// SIMATIC STEP 7 (V5.x) project ZEn01_11_STEP7__Com_SFC1
// program: ProgrammClient(MPI=10)
// program: ProgrammServer(MPI=12)
// program: ProgrammServer(MPI=15)

SYMBOL_TABLE
"Data_X_PUT"	DB 1	DB 1
"Data_X_GET"	DB 2	DB 2
"Data_X_SEND"	DB 3	DB 3
"Modify Values"	FC 1	FC 1
"Communication(send)"	FC 10	FC 10
"CYCL_EXC"	OB 1	OB 1	// Cycle Execution
"CYC_INT5"	OB 35	OB 35	// Cyclic Interrupt 5
"COMPLETE RESTART"	OB 100	OB 100	// Complete Restart
"X_SEND"	SFC 65	SFC 65
"X_RCV"	SFC 66	SFC 66
"X_GET"	SFC 67	SFC 67
"X_PUT"	SFC 68	SFC 68
"X_ABORT"	SFC 69	SFC 69
"I_GET"	SFC 72	SFC 72
"I_PUT"	SFC 73	SFC 73
"I_ABORT"	SFC 74	SFC 74
END_SYMBOL_TABLE

FUNCTION "Modify Values" : VOID	// FC 1
TITLE = Function for Generating a Modifiable Date
AUTHOR : SIEMENS
VERSION : 1.0
BEGIN
NETWORK
TITLE = Incrementing and Saving a Value
      L     MD 60;
      L     1;
      +D;
      T     MD 60;
      T     DB1.DBD 0;	//Save the variables to be sent in a double word
      T     DB3.DBD 0;
END_FUNCTION

FUNCTION "Communication(send)" : VOID	// FC 10
TITLE = Communicating with Both Servers
AUTHOR : SIEMENS
VERSION : 1.0
BEGIN
NETWORK
TITLE = Communicating with Server MPI 15
//Scan to see whether the SFCs X_PUT, X_GET, and X_SEND have communicated with 
//server MPI 15
      A     M 100.6;	//SFC X_PUT: Communication finished?
      A     M 101.6;	//SFC X_GET: Communication finished?
      A     M 102.6;	//SFC X_SEND: Communication finished?
      JC    net2;	//Jump to communication with server MPI 12
//                                        if the condtion is fulfilled. 
//Query which SFC is currently active?
      L     MW 50;	//SFC X_PUT active?
      L     1;
      ==I;
      JC    m001;	//Jump to SFC X_PUT
      L     MW 50;	//SFC X_GET active?
      L     2;
      ==I;
      JC    m002;	//Jump to SFC X_GET
      L     MW 50;	//SFC X_SEND active?
      L     3;
      ==I;
      JC    m003;	//Jump to SFC X_SEND
      BEU;
m001: CALL  "X_PUT" (
           REQ                      := M 100.2,
           CONT                     := M 100.3,
           DEST_ID                  := W#16#F,
           VAR_ADDR                 := "Data_X_PUT".Array10Bytes,
           SD                       := "Data_X_PUT".Array10Bytes,
           RET_VAL                  := MW 130,
           BUSY                     := M 100.4);	//Call X_PUT block / Transfer data (Yes/No)? / Maintain connection (Yes/No)? / Address of receiver / Address within communication partner / Send data 10 bytes (DB1) / Status display, negative if an error occurs / SFC active?
//Edge evaluation: Is communication with the falling edge of the BUSY bit
//finished?
      A     M 100.4;
      FN    M 100.5;
      S     M 100.6;	//Set memory bit: X_PUT is finished.
      JC    m004;	//Jump to increment the communication memory bit
      BEU;
m002: CALL  "X_GET" (
           REQ                      := M 101.2,
           CONT                     := M 101.3,
           DEST_ID                  := W#16#F,
           VAR_ADDR                 := "Data_X_GET".DoubleWord,
           RET_VAL                  := MW 132,
           BUSY                     := M 101.4,
           RD                       := "Data_X_GET".DoubleWord);	//Call X_SEND block / Transfer data (Yes/No)? / Maintain connection (Yes/No)? / Address of receiver / Address of variable in communication partner / Status display, negative if an error occurs / SFC active? / Pointer to address to which receive data are written
//Edge evaluation: Is communication with the falling edge of the BUSY bit
//finished?
      A     M 101.4;
      FN    M 101.5;
      S     M 101.6;	//Set memory bit: X_GET is finished.
      JC    m005;	//Jump to increment the communication counter
      BEU;
m003: CALL  "X_SEND" (
           REQ                      := M 102.2,
           CONT                     := M 102.3,
           DEST_ID                  := W#16#F,
           REQ_ID                   := DW#16#3,
           SD                       := "Data_X_SEND".Array3Words,
           RET_VAL                  := MW 134,
           BUSY                     := M 102.4);	//Call X_SEND block / Transfer data (Yes/No)? / Maintain connection (Yes/No)? / Address of receiver / Job number 3 / Send data 3 words (DB3) / Status display / SFC active?
//Edge evaluation: Is communication with the falling edge of the BUSY bit
//finished?
      A     M 102.4;
      FN    M 102.5;
      S     M 102.6;	//Set memory bit: X_SEND is finished.
      JC    m006;	//Jump to increment the communication counter
      BEU;
//In the following section, the communication counter is incremented following communication. 
m004: L     2;	//Increment on executing X_PUT
      T     MW 50;
      CALL  "Modify Values";	//The values in the variables are incremented
      BEU;
m005: L     3;	//Increment on executing X_GET
      T     MW 50;
      CALL  "Modify Values";	//The values in the variables are incremented
      BEU;
m006: L     1;	//Increment on executing X_SEND
      T     MW 50;
      CALL  "Modify Values";	//The values in the variables are incremented
NETWORK
TITLE = Communicating with Server MPI 12
//Query which SFC is currently active
net2: L     MW 52;	//SFC X_ABORT active?
      L     1;
      ==I;
      JC    m007;	//Jump to SFC X_ABORT
      L     MW 52;	//SFC X_SEND active?
      L     2;
      ==I;
      JC    m008;	//Jump to SFC X_SEND
      L     MW 52;	//SFC X_ABORT active?
      L     3;
      ==I;
      JC    m009;	//Jump to SFC X_ABORT
      BEU;
//In the following section of this network, the SFC X_ABORT is called to disconnect the 
//connection to the server MPI 15 which was established in network 1.
//The connection resource for SFC X_SEND in this network is available for this.
m007: CALL  "X_ABORT" (
           REQ                      := M 104.2,
           DEST_ID                  := W#16#F,
           RET_VAL                  := MW 136,
           BUSY                     := M 104.4);	//Call to abort connection to CPU-MPI 15 / Abort connection to CPU MPI address 15? / MPI address 15 / Return value of SFC / SFC active?
//Edge evaluation: Has the connection been aborted with the falling edge of the BUSY bit?
      A     M 104.4;
      FN    M 104.5;
      JC    m010;	//Jump to increment the communication memory word
      BEU;
//In the following section of this network, the SFC X_SEND is called to communicate 
//with the server MPI 12.
m008: CALL  "X_SEND" (
           REQ                      := M 105.2,
           CONT                     := M 105.3,
           DEST_ID                  := W#16#C,
           REQ_ID                   := DW#16#2,
           SD                       := "Data_X_PUT".Array10Bytes,
           RET_VAL                  := MW 138,
           BUSY                     := M 105.4);	//Call SFC X_SEND / Start data exchange? / Maintain connection following communication? / MPI address 12 / Job number 2 / Variable to be sent / Return value for error evaluation / SFC active?
//Edge evaluation: Is communication with the falling edge of the BUSY bit
//finished?
      A     M 105.4;
      FN    M 105.5;
      JC    m011;	//Jump to increment the communication memory word
      BEU;
//In the following section of this network, the SFC X_ABORT is called to disconnect the 
//connection to the server MPI 12 which was established in this network by SFC X_SEND.
//The connection resource for the SFCs in network 1 then becomes available again.
m009: CALL  "X_ABORT" (
           REQ                      := M 106.2,
           DEST_ID                  := W#16#C,
           RET_VAL                  := MW 140,
           BUSY                     := M 106.4);	//Call to abort connection to CPU MPI 12 / Abort connection to CPU MPI address 12? / MPI address 12
//Edge evaluation: Has the connection been aborted with the falling edge of the BUSY bit?
      A     M 106.4;
      FN    M 106.5;
      JC    m012;	//Jump to increment the communication memory word
      BEU;
//In the following section, the communication counter is incremented after an SFC has been 
//executed.
m010: L     2;	//Increment after executing X_ABORT with server MPI 15
      T     MW 52;
      BEU;
m011: L     3;	//Increment after executing X_SEND
      T     MW 52;
      BEU;
m012: L     1;	//Increment after executing X_ABORT with server MPI 12
      T     MW 52;
//Reset the memory bits in the first network: The SFC must have finished communicating 
//before the SFCs can be called again from the first network.
      CLR;
      =     M 100.6;	//Reset the memory bit: SFC X_PUT has been executed
      =     M 101.6;	//Reset the memory bit: SFC X_GET has been executed
      =     M 102.6;	//Reset the memory bit: SFC X_SEND has been executed
END_FUNCTION

DATA_BLOCK "Data_X_PUT"	// DB 1
AUTHOR : SIEMENS
VERSION : 1.0
  STRUCT
   Array10Bytes : ARRAY  [1 .. 10 ] OF //Array of 10 bytes
   BYTE  := 5 (B#16#10) , 5 (B#16#10) ;
  END_STRUCT ;	
BEGIN
   Array10Bytes[1] := B#16#10;
   Array10Bytes[2] := B#16#10;
   Array10Bytes[3] := B#16#10;
   Array10Bytes[4] := B#16#10;
   Array10Bytes[5] := B#16#10;
   Array10Bytes[6] := B#16#10;
   Array10Bytes[7] := B#16#10;
   Array10Bytes[8] := B#16#10;
   Array10Bytes[9] := B#16#10;
   Array10Bytes[10] := B#16#10;
END_DATA_BLOCK

DATA_BLOCK "Data_X_GET"	// DB 2
AUTHOR : SIEMENS
VERSION : 1.0
  STRUCT
   DoubleWord : DWORD  := DW#16#2D;	//Double word
  END_STRUCT ;	
BEGIN
   DoubleWord := DW#16#2D;
END_DATA_BLOCK

DATA_BLOCK "Data_X_SEND"	// DB 3
AUTHOR : SIEMENS
VERSION : 1.0
  STRUCT
   Array3Words : ARRAY  [1 .. 3 ] OF //Array of 3 words
   WORD  := 3 (W#16#3) ;
  END_STRUCT ;	
BEGIN
   Array3Words[1] := W#16#3;
   Array3Words[2] := W#16#3;
   Array3Words[3] := W#16#3;
END_DATA_BLOCK

ORGANIZATION_BLOCK "CYCL_EXC"	// OB 1
TITLE = Cyclically Processing Program
AUTHOR : SIEMENS
VERSION : 1.0
VAR_TEMP
  OB1_EV_CLASS : BYTE ;	//Bits 0 to 3 = 1 (incoming event), bits 4 to 7 = 1 (event class 1)
  OB1_SCAN_1 : BYTE ;	//1 (Cold restart scan 1 of OB1), 3 Scan 2-n of OB 1)
  OB1_PRIORITY : BYTE ;	//1 (Priority of 1 is lowest)
  OB1_OB_NUMBR : BYTE ;	//1 (Organization block 1, OB1)
  OB1_RESERVED_1 : BYTE ;	//Reserved for system
  OB1_RESERVED_2 : BYTE ;	//Reserved for system
  OB1_PREV_CYCLE : INT ;	//Cycle time of previous OB1 scan (milliseconds)
  OB1_MIN_CYCLE : INT ;	//Minimum cycle time of OB1 (milliseconds)
  OB1_MAX_CYCLE : INT ;	//Maximum cycle time of OB1 (milliseconds)
  OB1_DATE_TIME : DATE_AND_TIME ;	//Date and time OB1 started
END_VAR
BEGIN
NETWORK
TITLE = Default Settings of the SFC Parameters
//********************************************************************************
//********************
//General Description of the Communication Procedures of this Client CPU
//********************************************************************************
//********************
//
//Three variables are exchanged between this client station ("S7-300 Client MPI 
//10") and the two 
//server stations ("S7-300 Server MPI 12" and "S7-300 Server MPI 15").
//The variable "X_PUT-1".Feld10byte is sent to server MPI 15 with the SFC X_PUT 
//and to server MPI 10 
//with the SFC X_SEND. You only require one connection resource in order to 
//communicate with the two 
//different servers, because the connections are disconnected with the SFC 
//X_ABORT between communication  
//procedures. In this way, connection resources for communication with other MPI 
//subnet partners are 
//not occupied unnecessarily. The variable "X_GET-1".Doppelwort is read out from 
//the server MPI 15 
//with the SFC X_GET and stored in a variable of the same name in the client.
//The variable "X_SEND-1".Feld3Worte is written by the client to a variable of 
//the same name on the 
//server with the SFC X_SEND.
//The variables can be found in DBs 1 to 3 on both the client and the server 
//side. 
//The connection between the communicating CPUs is established the first time an 
//SFC is called
//and then maintained until the connection is disconnected and then established 
//again for 
//the next communication partner (only one connection resource is required).
//The SFCs are called by OB35 using a timer in order to make them independent of 
//the  
//scan cycle time of OB1 in the client and the server CPU.
//The timers for the OB calls are preset when the CPU is configured.
//In this CPU, OB35 is called every 100 ms (default), and this means that the 
//various SFCs are also 
//called every 100 ms (max.). 
//Once data exchange is complete, the data are changed in the variables in order 
//to show that  
//data have been received. If there is an error in the communication, and no data 
//are
//sent, the data in the receiver will not change. 
//If the receive data are continually changing, this means that data exchange is 
//taking place.
//
//Note:
//The memory words in which the RET_VALS of the SFCs are entered should be 
//evaluated while the  
//program is running. If an SFC registers an error value, the SFC calls which are 
//locked 
//in this example with the falling edge of the BUSY output may be correctly 
//executed. However,  
//no data will have been sent. If an SFC call is correctly executed and its 
//RET_VAL still 
//registers an error code, it is essential that you forward an error message to 
//this effect to 
//the user. As soon as the RET_VAL of an SFC becomes negative, this signals that 
//an error has
//occurred and that data may have been lost.
//
//Memory words in which the RET_VALs are entered:
//MW130, MW132, MW134, MW136, MW138, MW140
//
//The above note was not taken into account in this programming example, since 
//error messages 
//which may occur cannot be converted to corresponding messages (alarms which 
//appear on the device) 
//until a real control program is run.
NETWORK
TITLE = Presetting Communication
//By setting the following three memory bits, you can ensure that the connection 
//between 
//the communication partners is retained following each SFC call.
      SET;
      =     M 100.3;	//Connection should be maintained after SFC call 
      =     M 101.3;	//Connection should be maintained after SFC call
      =     M 102.3;	//Connection should be maintained after SFC call 
      =     M 105.3;	//Connection should be maintained after SFC call 
//Set start memory bit of SFC
      SET;
      =     M 100.2;	//SFC X_PUT 
      =     M 101.2;	//SFC X_GET
      =     M 102.2;	//SFC X_SEND
      =     M 104.2;	//SFC X_ABORT
      =     M 105.2;	//SFC X_SEND
      =     M 106.2;	//SFC X_ABORT
END_ORGANIZATION_BLOCK

ORGANIZATION_BLOCK "CYC_INT5"	// OB 35
TITLE = Block Call Timer-Controlled Every 100 ms
AUTHOR : SIEMENS
VERSION : 1.0
VAR_TEMP
  OB35_EV_CLASS : BYTE ;	//Bits 0 to 3 = 1 (incoming event), bits 4 to 7 = 1 (event class 1)
  OB35_STRT_INF : BYTE ;	//16#36 (OB35 has started)
  OB35_PRIORITY : BYTE ;	//11 (Priority of 1 is lowest)
  OB35_OB_NUMBR : BYTE ;	//35 (Organization block 35, OB35)
  OB35_RESERVED_1 : BYTE ;	//Reserved for system
  OB35_RESERVED_2 : BYTE ;	//Reserved for system
  OB35_PHASE_OFFSET : WORD ;	//Phase offset (ms)
  OB35_RESERVED_3 : INT ;	//Reserved for system
  OB35_EXC_FREQ : INT ;	//Frequency of execution (ms)
  OB35_DATE_TIME : DATE_AND_TIME ;	//Date and time OB35 started
END_VAR
BEGIN
NETWORK
TITLE =
      CALL  "Communication(send)";	//Call communication with servers
END_ORGANIZATION_BLOCK

ORGANIZATION_BLOCK "COMPLETE RESTART"	// OB 100
AUTHOR : SIEMENS
VERSION : 1.0
VAR_TEMP
  OB100_EV_CLASS : BYTE ;	//16#13, Event class 1, entering event state, event logged in diagnostic buffer
  OB100_STRTUP : BYTE ;	//16#81/82/83/84 Method of startup
  OB100_PRIORITY : BYTE ;	//27 (Priority of 1 is lowest)
  OB100_OB_NUMBR : BYTE ;	//100 (Organization block 100, OB100)
  OB100_RESERVED_1 : BYTE ;	//Reserved for system
  OB100_RESERVED_2 : BYTE ;	//Reserved for system
  OB100_STOP : WORD ;	//Event that caused CPU to stop (16#4xxx)
  OB100_STRT_INFO : DWORD ;	//Information on how system started
  OB100_DATE_TIME : DATE_AND_TIME ;	//Date and time OB100 started
END_VAR
BEGIN
NETWORK
TITLE = Initial Value Assignment
      L     1;	//Start value for communication counter
//Communication counter for data exchange with the station "S7-300 Server MPI 15" 
      T     MW 50;
//Communication counter for data exchange with the station "S7-300 Server MPI 12" 
      T     MW 52;
END_ORGANIZATION_BLOCK

SYMBOL_TABLE
"Communication(receive)"	FC 20	FC 20
"CYCL_EXC"	OB 1	OB 1	// Cycle Execution
"CYC_INT5"	OB 35	OB 35	// Cyclic Interrupt 5
"COMPLETE RESTART"	OB 100	OB 100	// Complete Restart
"X_SEND"	SFC 65	SFC 65
"X_RCV"	SFC 66	SFC 66
"X_GET"	SFC 67	SFC 67
"X_PUT"	SFC 68	SFC 68
"X_ABORT"	SFC 69	SFC 69
"I_GET"	SFC 72	SFC 72
"I_PUT"	SFC 73	SFC 73
"I_ABORT"	SFC 74	SFC 74
END_SYMBOL_TABLE

FUNCTION "Communication(receive)" : VOID	// FC 20
AUTHOR : SIEMENS
VERSION : 1.0
VAR_TEMP
  NIL_PTR : ANY ;	//NIL pointer, required in order to discard data
END_VAR
BEGIN
NETWORK
TITLE = Timer-Controlled Call of the X_RCV Block
//In this block, the SFC X_RCV is called every 10 ms using a timer.
//
//If the receive data are not evaluated for any reason, they must be 
//removed from the receive buffer and written to a NIL pointer.
//The following section of this network contains the branch instruction which
//determines whether the data are received or discarded.
//
      JU    add;	//Jump to accept the receive data
//    SPA   disc                        //Jump to discard the receive data
      BEU;
add:  SET;	//Set the accept memory bit
      =     M 100.2;
      CALL  "X_RCV" (
           EN_DT                    := M 100.2,
           RET_VAL                  := MW 132,
           REQ_ID                   := MD 120,
           NDA                      := M 101.5,
           RD                       := P#M 100.0 BYTE 10);	//Call receive SFC to accept the data / Accept data? / Return value / Job number / Receive new data? / Data area to which the receive data are added
NETWORK
TITLE = Discarding the Receive Data
//disc: NOP   1                         //This line must be included if the 
//receive data are to be 
//                                        discarded with the NIL pointer.
// (network holds code this reader does not know; not shown)
END_FUNCTION

ORGANIZATION_BLOCK "CYCL_EXC"	// OB 1
VERSION : 0.1
VAR_TEMP
  OB1_EV_CLASS : BYTE ;	//Bits 0-3 = 1 (Coming event), Bits 4-7 = 1 (Event class 1)
  OB1_SCAN_1 : BYTE ;	//1 (Cold restart scan 1 of OB 1), 3 (Scan 2-n of OB 1)
  OB1_PRIORITY : BYTE ;	//1 (Priority of 1 is lowest)
  OB1_OB_NUMBR : BYTE ;	//1 (Organization block 1, OB1)
  OB1_RESERVED_1 : BYTE ;	//Reserved for system
  OB1_RESERVED_2 : BYTE ;	//Reserved for system
  OB1_PREV_CYCLE : INT ;	//Cycle time of previous OB1 scan (milliseconds)
  OB1_MIN_CYCLE : INT ;	//Minimum cycle time of OB1 (milliseconds)
  OB1_MAX_CYCLE : INT ;	//Maximum cycle time of OB1 (milliseconds)
  OB1_DATE_TIME : DATE_AND_TIME ;	//Date and time OB1 started
END_VAR
BEGIN
// (block stored without names or comments; labels and parameter names are numbered)
END_ORGANIZATION_BLOCK

ORGANIZATION_BLOCK "CYC_INT5"	// OB 35
TITLE = Call Every 100 ms
AUTHOR : SIEMENS
VERSION : 1.0
VAR_TEMP
  OB35_EV_CLASS : BYTE ;	//Bits 0 to 3 = 1 (incoming event), bits 4 to 7 = 1 (event class 1)
  OB35_STRT_INF : BYTE ;	//16#36 (OB35 has started)
  OB35_PRIORITY : BYTE ;	//11 (Priority of 1 is lowest)
  OB35_OB_NUMBR : BYTE ;	//35 (Organization block 35, OB35)
  OB35_RESERVED_1 : BYTE ;	//Reserved for system
  OB35_RESERVED_2 : BYTE ;	//Reserved for system
  OB35_PHASE_OFFSET : WORD ;	//Phase offset (ms)
  OB35_RESERVED_3 : INT ;	//Reserved for system
  OB35_EXC_FREQ : INT ;	//Frequency of execution (ms)
  OB35_DATE_TIME : DATE_AND_TIME ;	//Date and time OB35 started
END_VAR
BEGIN
NETWORK
TITLE =
      CALL  "Communication(receive)";	//Call data receive function
END_ORGANIZATION_BLOCK

SYMBOL_TABLE
"Data_X_PUT-1"	DB 1	DB 1
"Data_X_GET-1"	DB 2	DB 2
"Data_X_SEND-1"	DB 3	DB 3
"Communication(receive)"	FC 30	FC 30
"CYCL_EXC"	OB 1	OB 1	// Cycle Execution
"CYC_INT5"	OB 35	OB 35	// Cyclic Interrupt 5
"COMPLETE RESTART"	OB 100	OB 100	// Complete Restart
"X_SEND"	SFC 65	SFC 65
"X_RCV"	SFC 66	SFC 66
"X_GET"	SFC 67	SFC 67
"X_PUT"	SFC 68	SFC 68
"X_ABORT"	SFC 69	SFC 69
"I_GET"	SFC 72	SFC 72
"I_PUT"	SFC 73	SFC 73
"I_ABORT"	SFC 74	SFC 74
END_SYMBOL_TABLE

FUNCTION "Communication(receive)" : VOID	// FC 30
AUTHOR : SIEMENS
VERSION : 1.0
VAR_TEMP
  NIL_PTR : ANY ;	//NIL pointer, required in order to discard data
END_VAR
BEGIN
NETWORK
TITLE = Timer-Controlled Call of SFC X_RCV
//Receiving an array of 3 words
//If the receive data are not evaluated for any reason, they must be 
//removed from the receive buffer and written to a NIL pointer.
//The following section of this network contains the branch instruction which
//determines whether the data are received or discarded.
//
      JU    add;	//Jump to accept the receive data
//    SPA   disc                        //Jump to discard the receive data
      BEU;
add:  SET;	//Set EN_DT to accept the receive data
      =     M 100.2;
      CALL  "X_RCV" (
           EN_DT                    := M 100.2,
           RET_VAL                  := MW 132,
           REQ_ID                   := MD 120,
           NDA                      := M 101.5,
           RD                       := "Data_X_SEND-1".Array3Words);	//Call SFC X_RCV / Add receive data to user memory?  / Return value / Job number of receive data / Have data been received? / Memory area to which the receive data are added
      BEU;
NETWORK
TITLE = Discarding the Receive Data
//disc: NOP   1                         //This line must be included if the 
//receive data are to be
//                                        discarded with the NIL pointer.
// (network holds code this reader does not know; not shown)
END_FUNCTION

DATA_BLOCK "Data_X_PUT-1"	// DB 1
AUTHOR : SIEMENS
VERSION : 1.0
  STRUCT
   Array10Byte : ARRAY  [1 .. 10 ] OF //Array of 10 bytes
   BYTE  := 5 (B#16#10) , 5 (B#16#10) ;
  END_STRUCT ;	
BEGIN
   Array10Byte[1] := B#16#10;
   Array10Byte[2] := B#16#10;
   Array10Byte[3] := B#16#10;
   Array10Byte[4] := B#16#10;
   Array10Byte[5] := B#16#10;
   Array10Byte[6] := B#16#10;
   Array10Byte[7] := B#16#10;
   Array10Byte[8] := B#16#10;
   Array10Byte[9] := B#16#10;
   Array10Byte[10] := B#16#10;
END_DATA_BLOCK

DATA_BLOCK "Data_X_GET-1"	// DB 2
AUTHOR : SIEMENS
VERSION : 1.0
  STRUCT
   DoubleWord : DWORD  := DW#16#2D;	//Double word
  END_STRUCT ;	
BEGIN
   DoubleWord := DW#16#2D;
END_DATA_BLOCK

DATA_BLOCK "Data_X_SEND-1"	// DB 3
AUTHOR : SIEMENS
VERSION : 1.0
  STRUCT
   Array3Words : ARRAY  [1 .. 3 ] OF //Array of 3 words
   WORD  := 3 (W#16#3) ;
  END_STRUCT ;	
BEGIN
   Array3Words[1] := W#16#3;
   Array3Words[2] := W#16#3;
   Array3Words[3] := W#16#3;
END_DATA_BLOCK

ORGANIZATION_BLOCK "CYCL_EXC"	// OB 1
VERSION : 0.1
VAR_TEMP
  OB1_EV_CLASS : BYTE ;	//Bits 0-3 = 1 (Coming event), Bits 4-7 = 1 (Event class 1)
  OB1_SCAN_1 : BYTE ;	//1 (Cold restart scan 1 of OB 1), 3 (Scan 2-n of OB 1)
  OB1_PRIORITY : BYTE ;	//1 (Priority of 1 is lowest)
  OB1_OB_NUMBR : BYTE ;	//1 (Organization block 1, OB1)
  OB1_RESERVED_1 : BYTE ;	//Reserved for system
  OB1_RESERVED_2 : BYTE ;	//Reserved for system
  OB1_PREV_CYCLE : INT ;	//Cycle time of previous OB1 scan (milliseconds)
  OB1_MIN_CYCLE : INT ;	//Minimum cycle time of OB1 (milliseconds)
  OB1_MAX_CYCLE : INT ;	//Maximum cycle time of OB1 (milliseconds)
  OB1_DATE_TIME : DATE_AND_TIME ;	//Date and time OB1 started
END_VAR
BEGIN
// (block stored without names or comments; labels and parameter names are numbered)
END_ORGANIZATION_BLOCK

ORGANIZATION_BLOCK "CYC_INT5"	// OB 35
TITLE = Call Every 100 ms
AUTHOR : SIEMENS
VERSION : 1.0
VAR_TEMP
  OB35_EV_CLASS : BYTE ;	//Bits 0 to 3 = 1 (incoming event), bits 4 to 7 = 1 (event class 1)
  OB35_STRT_INF : BYTE ;	//16#36 (OB35 has started)
  OB35_PRIORITY : BYTE ;	//11 (Priority of 1 is lowest)
  OB35_OB_NUMBR : BYTE ;	//35 (Organization block 35, OB35)
  OB35_RESERVED_1 : BYTE ;	//Reserved for system
  OB35_RESERVED_2 : BYTE ;	//Reserved for system
  OB35_PHASE_OFFSET : WORD ;	//Phase offset (ms)
  OB35_RESERVED_3 : INT ;	//Reserved for system
  OB35_EXC_FREQ : INT ;	//Frequency of execution (ms)
  OB35_DATE_TIME : DATE_AND_TIME ;	//Date and time OB35 started
END_VAR
BEGIN
NETWORK
TITLE =
      CALL  "Communication(receive)";	//Call data receive function
END_ORGANIZATION_BLOCK

ORGANIZATION_BLOCK "COMPLETE RESTART"	// OB 100
AUTHOR : SIEMENS
VERSION : 1.0
VAR_TEMP
  OB100_EV_CLASS : BYTE ;	//16#13, Event class 1, entering event state, event logged in diagnostic buffer
  OB100_STRTUP : BYTE ;	//16#81/82/83/84 Method of startup
  OB100_PRIORITY : BYTE ;	//27 (Priority of 1 is lowest)
  OB100_OB_NUMBR : BYTE ;	//100 (Organization block 100, OB100)
  OB100_RESERVED_1 : BYTE ;	//Reserved for system
  OB100_RESERVED_2 : BYTE ;	//Reserved for system
  OB100_STOP : WORD ;	//Event that caused CPU to stop (16#4xxx)
  OB100_STRT_INFO : DWORD ;	//Information on how system started
  OB100_DATE_TIME : DATE_AND_TIME ;	//Date and time OB100 started
END_VAR
BEGIN
NETWORK
TITLE = Start Settings
//Load ASCII characters to MD50 and MD54
      L     'OTTO';
      T     MD 50;
      L     'HANS';
      T     MD 54;
//Preset counter
      L     0;
      T     MW 58;
END_ORGANIZATION_BLOCK
